# EPICS autosave request: GALILMUL/iocBoot/iocGALILMUL-IOC-02/GALILMUL_02_positions_norestore.req
file "GALIL_controller_positions.req" "P=$(P),CCP=$(MTRCTRL1)"
file "GALIL_controller_positions.req" "P=$(P),CCP=$(MTRCTRL2)"
